(* PLC project EtherlabMaster SDO Blocks, EtherlabMaster EtherlabMaster 1 *)
(* stored: creationDateTime 2012-10-22T12:12:45, modificationDateTime 2012-11-13T18:03:39 *)

FUNCTION_BLOCK EtherLabSDOUpload
  VAR_INPUT
    EXECUTE : BOOL;
    POS : INT;
    INDEX : UINT;
    SUBINDEX : USINT;
    VARTYPE : STRING;
  END_VAR
  VAR_OUTPUT
    ACK : BOOL;
    VALID : BOOL;
    VALUE : STRING;
  END_VAR
  VAR
    PY0 : python_eval;
    PY1 : python_eval;
    EXECUTE0 : BOOL;
    STATE : INT := 0;
  END_VAR

{extern int AcquireSDOLock();}
{extern int HasAnswer();}
{extern void ReleaseSDOLock();}
CASE STATE OF
  0:
    IF EXECUTE AND NOT EXECUTE0 THEN
      STATE := 1;
      ACK := 0;
      VALID := 0;
      VALUE := 'None';
    END_IF;
  1:
    {if (AcquireSDOLock()) __SET_VAR(data__->,STATE, 2)}
  2:
    IF PY0.ACK THEN
      STATE := 3;
    END_IF;
  3:
    {if (HasAnswer()) __SET_VAR(data__->,STATE, 4)}
  4:
    IF PY1.ACK THEN
      ACK := 1;
      VALUE := PY1.RESULT;
      VALID := NE(VALUE, 'None');
      STATE := 0;
      {ReleaseSDOLock();}
    END_IF;
ELSE
  STATE := 0;
END_CASE;

EXECUTE0 := EXECUTE;
PY0(TRIG := STATE = 2, 
    CODE := CONCAT('EthercatSDOUpload(',
                   INT_TO_STRING(POS),
                   ',',
                   UINT_TO_STRING(INDEX),
                   ',',
                   USINT_TO_STRING(SUBINDEX),
                   ',"',
                   VARTYPE,
                   '")'));
PY1(TRIG := STATE = 4, 
    CODE := 'GetResult()');

          
END_FUNCTION_BLOCK

FUNCTION_BLOCK EtherLabSDODownload
  VAR_INPUT
    EXECUTE : BOOL;
    POS : INT;
    INDEX : UINT;
    SUBINDEX : USINT;
    VARTYPE : STRING;
    VALUE : STRING;
  END_VAR
  VAR_OUTPUT
    ACK : BOOL;
    ERROR : BOOL;
  END_VAR
  VAR
    PY0 : python_eval;
    PY1 : python_eval;
    EXECUTE0 : BOOL;
    STATE : INT := 0;
  END_VAR

{extern int AcquireSDOLock();}
{extern int HasAnswer();}
{extern void ReleaseSDOLock();}
CASE STATE OF
  0:
    IF EXECUTE AND NOT EXECUTE0 THEN
      STATE := 1;
      ACK := 0;
      ERROR := 0;
    END_IF;
  1:
    {if (AcquireSDOLock()) __SET_VAR(data__->,STATE, 2)}
  2:
    IF PY0.ACK THEN
      STATE := 3;
    END_IF;
  3:
    {if (HasAnswer()) __SET_VAR(data__->,STATE, 4)}
  4:
    IF PY1.ACK THEN
      ACK := 1;
      ERROR := EQ(PY1.RESULT, 'False');
      STATE := 0;
      {ReleaseSDOLock();}
    END_IF;
ELSE
  STATE := 0;
END_CASE;
EXECUTE0 := EXECUTE;
PY0(TRIG := STATE = 2, 
    CODE := CONCAT('EthercatSDODownload(',
                   INT_TO_STRING(POS),
                   ',',
                   UINT_TO_STRING(INDEX),
                   ',',
                   USINT_TO_STRING(SUBINDEX),
                   ',"',
                   VARTYPE,
                   '",',
                   VALUE,
                   ')'));
PY1(TRIG := STATE = 4, 
    CODE := 'GetResult()');

          
END_FUNCTION_BLOCK

FUNCTION_BLOCK EtherLabSetTorqueLimit
  VAR_INPUT
    Pos : INT;
    Execute : BOOL;
    TorqueLimitPos : UINT;
    TorqueLimitNeg : UINT;
  END_VAR
  VAR_OUTPUT
    Done : BOOL;
    Busy : BOOL;
    Error : BOOL;
    ErrorID : WORD;
  END_VAR
  VAR
    EtherLabSDOUpload0 : EtherLabSDODownload;
    EtherLabSDOUpload1 : EtherLabSDODownload;
    RS0 : RS;
  END_VAR
  VAR  (* added by the conversion: wires and edge detectors of the diagram *)
    _AND16_OUT : BOOL;
  END_VAR

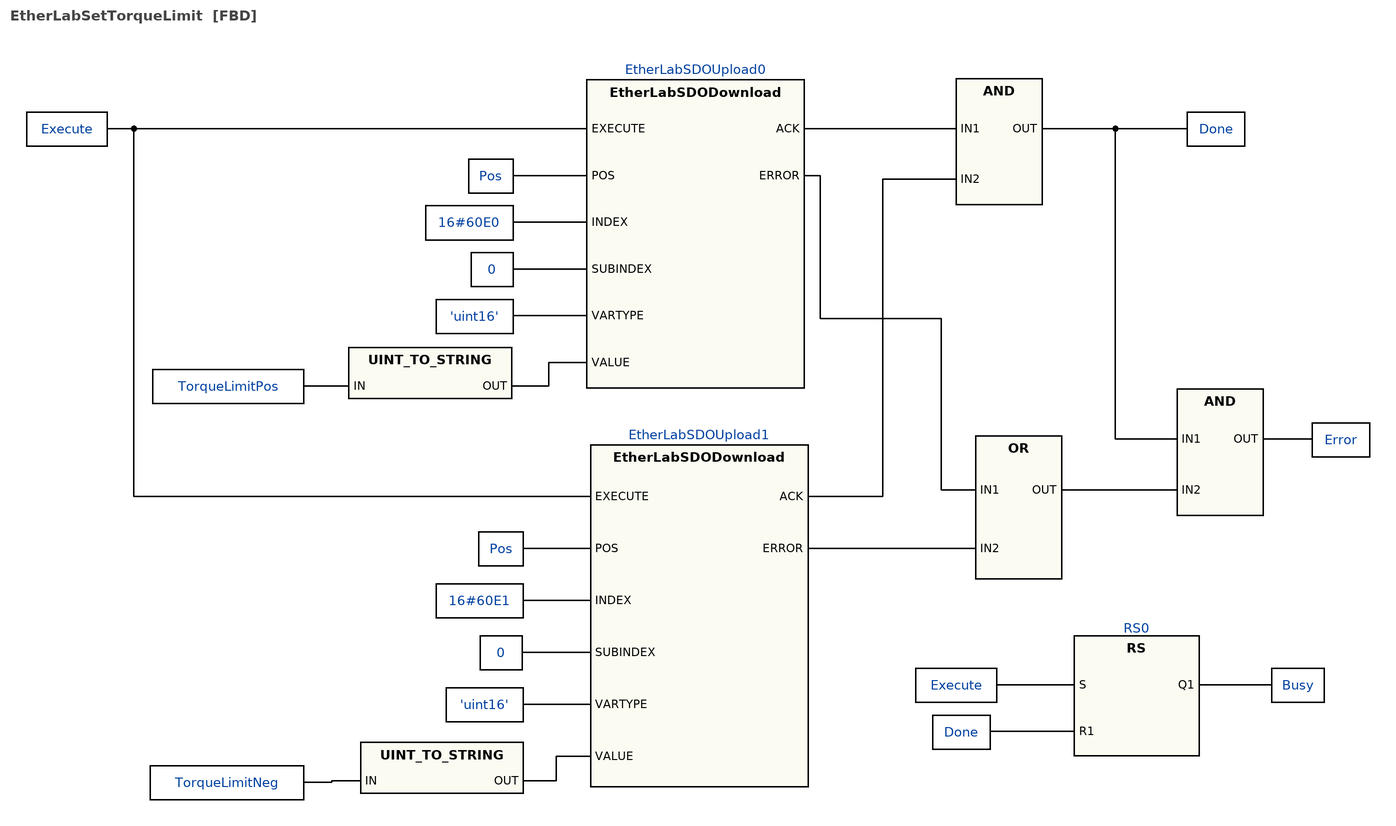
(* FBD diagram, written out as Structured Text *)
EtherLabSDOUpload0(EXECUTE := Execute, POS := Pos, INDEX := 16#60E0, SUBINDEX := 0, VARTYPE := 'uint16', VALUE := UINT_TO_STRING(TorqueLimitPos));
EtherLabSDOUpload1(EXECUTE := Execute, POS := Pos, INDEX := 16#60E1, SUBINDEX := 0, VARTYPE := 'uint16', VALUE := UINT_TO_STRING(TorqueLimitNeg));
_AND16_OUT := EtherLabSDOUpload0.ACK AND EtherLabSDOUpload1.ACK;
Done := _AND16_OUT;
Error := _AND16_OUT AND (EtherLabSDOUpload0.ERROR OR EtherLabSDOUpload1.ERROR);
RS0(S := Execute, R1 := Done);
Busy := RS0.Q1;
END_FUNCTION_BLOCK

FUNCTION_BLOCK EtherLabGetTorqueLimit
  VAR_INPUT
    Pos : INT;
    Execute : BOOL;
  END_VAR
  VAR_OUTPUT
    Done : BOOL;
    Busy : BOOL;
    Error : BOOL;
    ErrorID : WORD;
    TorqueLimitPos : UINT;
    TorqueLimitNeg : UINT;
  END_VAR
  VAR
    EtherLabSDOUpload0 : EtherLabSDOUpload;
    EtherLabSDOUpload1 : EtherLabSDOUpload;
    RS0 : RS;
  END_VAR
  VAR  (* added by the conversion: wires and edge detectors of the diagram *)
    _AND16_OUT : BOOL;
  END_VAR

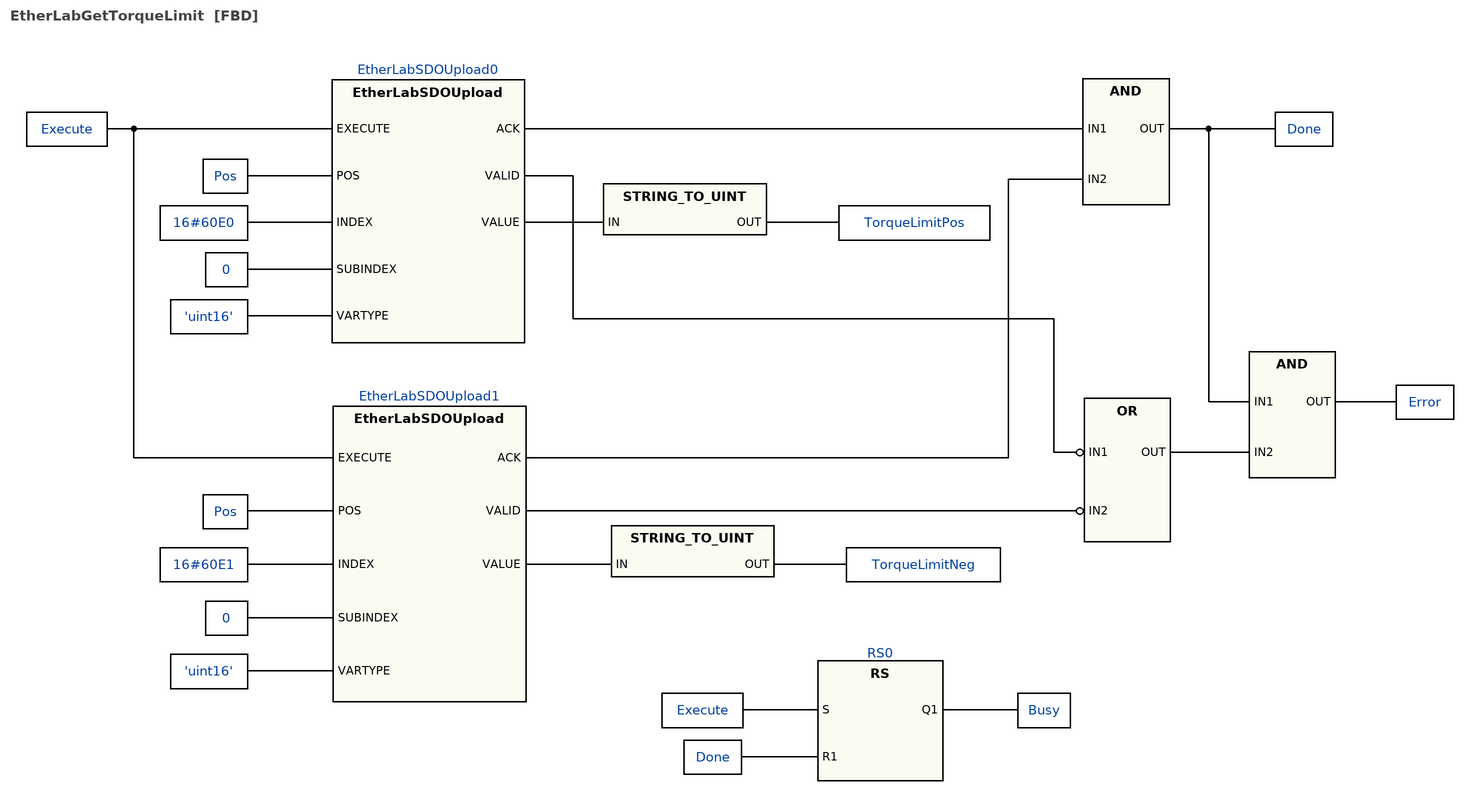
(* FBD diagram, written out as Structured Text *)
EtherLabSDOUpload0(EXECUTE := Execute, POS := Pos, INDEX := 16#60E0, SUBINDEX := 0, VARTYPE := 'uint16');
EtherLabSDOUpload1(EXECUTE := Execute, POS := Pos, INDEX := 16#60E1, SUBINDEX := 0, VARTYPE := 'uint16');
_AND16_OUT := EtherLabSDOUpload0.ACK AND EtherLabSDOUpload1.ACK;
Done := _AND16_OUT;
TorqueLimitPos := STRING_TO_UINT(EtherLabSDOUpload0.VALUE);
Error := _AND16_OUT AND (NOT EtherLabSDOUpload0.VALID OR NOT EtherLabSDOUpload1.VALID);
TorqueLimitNeg := STRING_TO_UINT(EtherLabSDOUpload1.VALUE);
RS0(S := Execute, R1 := Done);
Busy := RS0.Q1;
END_FUNCTION_BLOCK
